// TwinCAT 3 PLC project PLC
// ProgramVersion: 3.1.4023.0
// libraries:
//   Tc2_Standard, * (Beckhoff Automation GmbH)
//   Tc2_System, * (Beckhoff Automation GmbH)
//   Tc3_Module, * (Beckhoff Automation GmbH)
// project tree:
//   DUTs/ ST_Coordinate.TcDUT, ST_Food.TcDUT, ST_SnakePart.TcDUT
//   GVLs/ GVL_Constants.TcGVL, GVL_Variables.TcGVL
//   / PlcTask.TcTTO
//   POUs/ FB_Draw.TcPOU, FB_Food.TcPOU, GameEngine.TcPOU, FB_Snake.TcPOU, MAIN.TcPOU
// real-time tasks:
//   TASK PlcTask: cycle T#10ms, priority 20, ADS port 350

CONFIGURATION PLC
    RESOURCE PLC ON TwinCAT3
        TASK PlcTask(INTERVAL := T#10ms, PRIORITY := 20);
        PROGRAM MAIN WITH PlcTask : MAIN;
    END_RESOURCE
END_CONFIGURATION

// ---- DUTs/ST_Coordinate.TcDUT
TYPE ST_Coordinate :
STRUCT
	iColumnCoordinate 	: INT;
	iRowCoordinate	 	: INT;
END_STRUCT
END_TYPE

// ---- DUTs/ST_Food.TcDUT
TYPE ST_Food :
STRUCT
	stFoodCoordinate : ST_Coordinate;
END_STRUCT
END_TYPE

// ---- DUTs/ST_SnakePart.TcDUT
TYPE ST_SnakePart :
STRUCT
	stBodyCoordinate : ST_Coordinate;
END_STRUCT
END_TYPE

// ---- GVLs/GVL_Constants.TcGVL
{attribute 'qualified_only'}
VAR_GLOBAL CONSTANT
	SNAKE_LENGTH : INT := 10;
END_VAR

// ---- GVLs/GVL_Variables.TcGVL
{attribute 'qualified_only'}
VAR_GLOBAL 
	aStSnakeBody		: ARRAY[1..GVL_Constants.SNAKE_LENGTH] OF ST_SnakePart;
	aStSnakeBodyEmpty	: ARRAY[1..GVL_Constants.SNAKE_LENGTH] OF ST_SnakePart;
	iSnakeLength		: INT;
	iSnakeDirection 	: INT;
	bDraw				: BOOL;
	bInit				: BOOL := FALSE;
	
	bGameOver			: BOOL;
	stFood				: ST_Food;
END_VAR

// ---- POUs/MAIN.TcPOU
PROGRAM MAIN
VAR
	
END_VAR

GameEngine();

END_PROGRAM

// ---- POUs/GameEngine.TcPOU
PROGRAM GameEngine
VAR
	fbSnake			: FB_Snake;
	fbFood			: FB_Food;
	fbDraw			: FB_Draw;
	
	updateTimer		: TON;
	bSnakeMove		: BOOL;

	rTrig			: R_TRIG;
END_VAR

rTrig(CLK := GVL_Variables.bInit);
fbSnake(aStSnakeBody:= GVL_Variables.aStSnakeBody, iSnakeLength := GVL_Variables.iSnakeLength);
fbFood(stFood => GVL_Variables.stFood);

IF rTrig.Q THEN
	GVL_Variables.aStSnakeBody := GVL_Variables.aStSnakeBodyEmpty;
	GVL_Variables.aStSnakeBody[1].stBodyCoordinate.iColumnCoordinate := 5;
	GVL_Variables.aStSnakeBody[1].stBodyCoordinate.iRowCoordinate := 5;
	GVL_Variables.iSnakeLength := 1;
	GVL_Variables.bGameOver := FALSE;
	GVL_Variables.bInit := FALSE;
END_IF

IF NOT GVL_Variables.bGameOver THEN
	updateTimer(IN := NOT updateTimer.Q, PT := T#1S);
	IF updateTimer.Q THEN
		bSnakeMove := fbSnake.M_Move(GVL_Variables.iSnakeDirection);		
	END_IF

	IF fbSnake.M_Die() THEN
		GVL_Variables.bGameOver := TRUE;
	END_IF

	IF fbSnake.M_Eat(GVL_Variables.stFood) THEN
		fbFood.M_Generate();
	END_IF
END_IF

fbDraw();
GVL_Variables.bDraw := fbDraw.M_Draw();

END_PROGRAM

// ---- POUs/FB_Snake.TcPOU
FUNCTION_BLOCK FB_Snake
VAR_IN_OUT
	//first item is head
	aStSnakeBody	: ARRAY[1..GVL_Constants.SNAKE_LENGTH] OF ST_SnakePart;
	iSnakeLength 	: INT;
END_VAR
VAR_OUTPUT
END_VAR
VAR
	
END_VAR

METHOD M_Die : BOOL
VAR_INPUT
END_VAR

VAR
	iPartIndex: INT;
END_VAR
{warning disable C0371}
IF NOT __ISVALIDREF(aStSnakeBody) AND NOT __ISVALIDREF(iSnakeLength) THEN
     RETURN;
END_IF

M_Die := FALSE;
IF aStSnakeBody[1].stBodyCoordinate.iColumnCoordinate > 9 OR aStSnakeBody[1].stBodyCoordinate.iColumnCoordinate < 0 OR
	aStSnakeBody[1].stBodyCoordinate.iRowCoordinate < 0 OR aStSnakeBody[1].stBodyCoordinate.iRowCoordinate > 9 THEN
	M_Die := TRUE;
END_IF

IF iSnakeLength >= 4 THEN
	FOR iPartIndex := iSnakeLength TO 2 BY -1 DO
		IF aStSnakeBody[1].stBodyCoordinate.iColumnCoordinate = aStSnakeBody[iPartIndex].stBodyCoordinate.iColumnCoordinate AND
			aStSnakeBody[1].stBodyCoordinate.iRowCoordinate = aStSnakeBody[iPartIndex].stBodyCoordinate.iRowCoordinate THEN
			M_Die := TRUE;
		END_IF
	END_FOR
END_IF

{warning restore C0371}
END_METHOD

//if head cordinate and food cordinate match then snake has eaten the food and got larger
METHOD PUBLIC M_Eat : BOOL
VAR_INPUT
	stFood		: ST_Food;
END_VAR
VAR
	bHasEaten	: BOOL;
END_VAR
{warning disable C0371}
IF NOT __ISVALIDREF(aStSnakeBody) AND NOT __ISVALIDREF(iSnakeLength) THEN
     RETURN;
END_IF

IF aStSnakeBody[1].stBodyCoordinate.iColumnCoordinate = stFood.stFoodCoordinate.iColumnCoordinate AND
	aStSnakeBody[1].stBodyCoordinate.iRowCoordinate = stFood.stFoodCoordinate.iRowCoordinate THEN	
	bHasEaten := TRUE;
ELSE
	bHasEaten := FALSE;
END_IF

IF bHasEaten AND iSnakeLength <= GVL_Constants.SNAKE_LENGTH THEN
	iSnakeLength := iSnakeLength + 1;
END_IF

M_Eat := bHasEaten;
{warning restore C0371}
END_METHOD

METHOD PUBLIC M_Move : BOOL
VAR_INPUT
	iHeadDirection : INT;
END_VAR

VAR
	bMoved			: BOOL;
	iPartIndex		: INT;
END_VAR
{warning disable C0371}
M_Move := FALSE;
IF NOT __ISVALIDREF(THIS^.aStSnakeBody) AND NOT __ISVALIDREF(iSnakeLength) THEN
     RETURN;
END_IF

FOR iPartIndex := iSnakeLength+1 TO 2 BY -1 DO
	aStSnakeBody[iPartIndex].stBodyCoordinate := aStSnakeBody[iPartIndex - 1].stBodyCoordinate;
END_FOR

IF iHeadDirection = 1 THEN	
	bMoved	:= TRUE;
	aStSnakeBody[1].stBodyCoordinate.iColumnCoordinate	:= aStSnakeBody[1].stBodyCoordinate.iColumnCoordinate - 1;
ELSIF iHeadDirection = 4  THEN
	bMoved	:= TRUE;
	aStSnakeBody[1].stBodyCoordinate.iColumnCoordinate := aStSnakeBody[1].stBodyCoordinate.iColumnCoordinate + 1;
ELSIF iHeadDirection = 3  THEN
	bMoved	:= TRUE;
	aStSnakeBody[1].stBodyCoordinate.iRowCoordinate	:=  aStSnakeBody[1].stBodyCoordinate.iRowCoordinate + 1;
ELSIF iHeadDirection = 2 THEN
	bMoved	:= TRUE;
	aStSnakeBody[1].stBodyCoordinate.iRowCoordinate	:= aStSnakeBody[1].stBodyCoordinate.iRowCoordinate - 1;
END_IF
M_Move := bMoved;
{warning restore C0371}
END_METHOD

END_FUNCTION_BLOCK

// ---- POUs/FB_Food.TcPOU
FUNCTION_BLOCK FB_Food
VAR_OUTPUT
	stFood 				: ST_Food;
END_VAR
VAR
	randomColumnNumGenerator :	DRAND;
	randomRowNumGenerator 	:	DRAND;
	iRandColumn				:	INT;
 	iRandRow				:	INT;
END_VAR

randomColumnNumGenerator(Seed:= iRandColumn+10);
randomRowNumGenerator(Seed:= iRandRow);

iRandColumn := LREAL_TO_INT(randomColumnNumGenerator.Num * 9);
iRandRow 	:= LREAL_TO_INT(randomRowNumGenerator.Num * 9);

METHOD M_Generate : BOOL;
VAR_INPUT
	
END_VAR
M_Generate := FALSE;
	stFood.stFoodCoordinate.iColumnCoordinate := iRandColumn; 
	stFood.stFoodCoordinate.iRowCoordinate := iRandRow; 
M_Generate := TRUE;
END_METHOD

END_FUNCTION_BLOCK

// ---- POUs/FB_Draw.TcPOU
FUNCTION_BLOCK FB_Draw
VAR
	bDraw			: BOOL;
 	OnTimer 		: TON;
	OffTimer 		: TON;
END_VAR

OnTimer(IN := NOT OffTimer.Q , PT := T#500MS);
OffTimer(IN := OnTimer.Q , PT := T#500ms);
bDraw := OnTimer.Q;

METHOD M_Draw : BOOL
VAR_INPUT
END_VAR
M_Draw := THIS^.bDraw;
END_METHOD

END_FUNCTION_BLOCK
